// TIA Portal V19 export
TYPE "MES_Msg"
// stored: Access Published
   STRUCT
      Id : DInt;   // Identificativo progressivo del messaggio log
      timestamp : String;   // Formato YYYY-MM-DD HH:MM:SS.mmm
      topic : UDInt;   // Codice argomento del log
      payLoad : String;   // Descriione dell' evento
   END_STRUCT;
END_TYPE
